(* IEC 61131-3 sources: CodesysTest/export/UN00 - Sharp Bagger/EM02 - Discharge/EM02_Discharge.pou/OKToFeedBag.prop, 1 file *)

(* ---- Get.pm.st ---- *)
(*#-#-#-#-#-#-#-#-#-#---Declaration---#-#-#-#-#-#-#-#-#-#-#-#-#*)

VAR
END_VAR
(*#-#-#-#-#-#-#-#-#-#---Implementation---#-#-#-#-#-#-#-#-#-#-#-#-#*)

OKToFeedBag := TRUE;
